Staubli VAL3: push_front.pgx

public program push_front(bool& x_res, MotionBuffer& x_cmd)
begin
end
